TYPE ST_CAMERA_TriggerID :
STRUCT
	nTriggerID			: UDINT;
	nScanNo				: INT := 1;
	nScannerIndex		: INT := 1;
END_STRUCT
END_TYPE

(* stored: Version 1.1.0.1
   DUT ST_CAMERA_TriggerID: Id {3a3747a6-78b4-43d9-9fb2-8764e0936882} *)
